Fanuc KAREL source: kt00904.KL

-- PROVISIONAL review KL for V1013-1; original PC SHA256 22d188b5745e1bc0054730e07e3409adb3e102d90dae7329e4e7de86137241d1
-- Incomplete behavior may be omitted. Consult companion uncertainty JSON. Do not deploy.
PROGRAM KT00904
%NOLOCKGROUP
BEGIN
  -- UNRESOLVED_PC offsets 5-20; opcodes 2E,22,32,35
  -- UNRESOLVED_PC offsets 25-40; opcodes 2E,22,32,35
  -- UNRESOLVED_PC offsets 45-60; opcodes 2E,22,32,35
  -- UNRESOLVED_PC offsets 65-80; opcodes 2E,22,32,35
  -- UNRESOLVED_PC offsets 85-111; opcodes 27,27,49,7E,AD,31,4A
  -- UNRESOLVED_PC offsets 116-120; opcodes 7F
END KT00904
